(* PLC project CookiePLC, Unknown Unnamed 1 *)
(* stored: creationDateTime 2025-02-05T12:34:47, modificationDateTime 2025-11-16T22:54:03 *)

FUNCTION_BLOCK mixer_rpm_function
  VAR_OUTPUT
    output_rpm : WORD;
  END_VAR
  VAR_INPUT
    valve_status : BOOL;
    hopper_weight : REAL;
    mixer_status : BOOL;
  END_VAR
  VAR
    noise : INT;
  END_VAR
  VAR_IN_OUT
    counter : INT;
  END_VAR

            counter := counter + 1;
IF counter > 10000 THEN
  counter := 0;
END_IF;

noise := counter MOD 2;

IF hopper_weight = 0.0 AND mixer_status = 1 THEN
  output_rpm := INT_TO_WORD(70 + noise);
ELSIF hopper_weight > 0.0 AND mixer_status = 1 AND valve_status = 1 THEN
  output_rpm := INT_TO_WORD(35 + noise);
ELSE
  output_rpm := INT_TO_WORD(0);
END_IF;
          
END_FUNCTION_BLOCK

FUNCTION_BLOCK vacuum_rpm_function
  VAR_INPUT
    input_rpm : WORD;
    vacuum_status : BOOL;
  END_VAR
  VAR_OUTPUT
    output_rpm : WORD;
  END_VAR
  VAR_INPUT
    max_rpm : WORD;
    manual : BOOL := 0;
    dv : BOOL;
  END_VAR
  VAR
    noise : INT;
  END_VAR
  VAR_IN_OUT
    counter : INT;
  END_VAR

            counter := counter + 1;
IF counter > 10000 THEN
  counter := 0;
END_IF;

noise := counter MOD 5;

IF NOT vacuum_status THEN
  output_rpm := 0;
ELSIF input_rpm > max_rpm THEN
  output_rpm := INT_TO_WORD(WORD_TO_INT(max_rpm) + noise);
ELSIF dv = 1 AND manual = 0 THEN
  output_rpm := INT_TO_WORD(1380 + noise);
ELSIF dv = 0 AND manual = 0 THEN
  output_rpm := INT_TO_WORD(1980 + noise);
ELSE
  IF (counter MOD 2) = 1 THEN
    output_rpm := INT_TO_WORD(WORD_TO_INT(input_rpm) + noise);
  ELSE
    output_rpm := INT_TO_WORD(WORD_TO_INT(input_rpm) - noise);
    END_IF;
END_IF;
          
END_FUNCTION_BLOCK

FUNCTION_BLOCK real_to_words
  VAR_INPUT
    Input : REAL;
  END_VAR
  VAR_OUTPUT
    High : WORD;
    Low : WORD;
  END_VAR

            {
    IEC_REAL var_in;
    IEC_WORD var_out[2];
    
    var_in = GetFbVar(INPUT);
    memcpy(var_out, &var_in, sizeof(var_in));
    SetFbVar(HIGH, var_out[0]);
    SetFbVar(LOW, var_out[1]);
}
    
    
          
END_FUNCTION_BLOCK

FUNCTION_BLOCK words_to_real
  VAR_INPUT
    High : WORD;
    Low : WORD;
  END_VAR
  VAR_OUTPUT
    Result : REAL;
  END_VAR

            {
    IEC_WORD var_in[2];

    IEC_REAL var_out;

    var_in[0] = GetFbVar(HIGH);

    var_in[1] = GetFbVar(LOW);

    memcpy(&var_out, var_in, sizeof(var_out));

    SetFbVar(RESULT, var_out);
}
          
END_FUNCTION_BLOCK

FUNCTION_BLOCK conveyor_fpm_function
  VAR_INPUT
    wirecut_cpm : WORD;
    cookie_margin : REAL;
    cookie_diameter : REAL;
  END_VAR
  VAR_OUTPUT
    conveyor_fpm : REAL;
  END_VAR

            conveyor_fpm := (WORD_TO_REAL(wirecut_cpm) * (cookie_margin+cookie_diameter)) / 12.0;
          
END_FUNCTION_BLOCK

FUNCTION_BLOCK flour_alarm_check
  VAR_INPUT
    Flour_weight : REAL;
  END_VAR
  VAR_OUTPUT
    Alarm : BOOL := FALSE;
  END_VAR

            IF Flour_weight <= 100.0 THEN
  Alarm := TRUE;
ELSE
  Alarm := FALSE;
END_IF;

          
END_FUNCTION_BLOCK

FUNCTION_BLOCK hopper_alarm_check
  VAR_INPUT
    Hopper_weight : REAL;
  END_VAR
  VAR_OUTPUT
    Alarm : BOOL := FALSE;
  END_VAR

            IF Hopper_weight <= 10.0 THEN
  Alarm := TRUE;
ELSE
  Alarm := FALSE;
END_IF;

          
END_FUNCTION_BLOCK

FUNCTION_BLOCK papercutter_cpm_function
  VAR
    rows : REAL;
  END_VAR
  VAR_INPUT
    paper_cutter : BOOL;
    cookie_diameter : REAL;
    cookie_margin : REAL;
    conveyor_fpm : REAL;
  END_VAR
  VAR
    float_cpm : REAL;
  END_VAR
  VAR_OUTPUT
    papercut_cpm : WORD;
  END_VAR

            
IF paper_cutter THEN
  rows := 5.0;
  float_cpm := (conveyor_fpm * 12.0) / (rows * (cookie_diameter+cookie_margin));
  papercut_cpm := REAL_TO_WORD(float_cpm);
ELSE
  papercut_cpm := 0;
END_IF;
          
END_FUNCTION_BLOCK

FUNCTION_BLOCK sugar_alarm_check
  VAR_INPUT
    Sugar_weight : REAL;
  END_VAR
  VAR_OUTPUT
    Alarm : BOOL := FALSE;
  END_VAR

            IF Sugar_weight <= 100.0 THEN
  Alarm := TRUE;
ELSE
  Alarm := FALSE;
END_IF;

          
END_FUNCTION_BLOCK

FUNCTION_BLOCK vacuum_alarm_rpm
  VAR_INPUT
    Dv : BOOL;
  END_VAR
  VAR_OUTPUT
    Cfm : REAL;
  END_VAR
  VAR_INPUT
    Vacuum_rpm : WORD;
  END_VAR
  VAR_OUTPUT
    Alarm : BOOL := FALSE;
  END_VAR

            

Cfm := ((-1.275 * 0.0000001) * (WORD_TO_REAL(Vacuum_rpm) * WORD_TO_REAL(Vacuum_rpm)) + (0.7896 * WORD_TO_REAL(Vacuum_rpm)) - 365.43);

IF Dv = 1 AND Cfm < 687.0 THEN 
  Alarm := TRUE;
ELSIF Dv = 0 AND Cfm < 1178.0 THEN
  Alarm := TRUE;
ELSE
  Alarm := FALSE;
END_IF;
  
          
END_FUNCTION_BLOCK

FUNCTION_BLOCK wirecut_cpm_function
  VAR_IN_OUT
    wirecut_cpm : WORD;
  END_VAR
  VAR_INPUT
    wirecutter : BOOL;
  END_VAR

            IF wirecutter THEN
  wirecut_cpm := 200;
ELSE
  wirecut_cpm := 0;
END_IF;
          
END_FUNCTION_BLOCK

PROGRAM tag_display
  VAR
    lcs_1_low AT %QW100 : WORD;  (* Load cell 1 for sugar (lower integer) *)
    lcs_1_high AT %QW101 : WORD;  (* Load cell 1 for sugar (higher integer) *)
    lcs_2_low AT %QW102 : WORD;  (* Load cell 2 for sugar (lower integer) *)
    lcs_2_high AT %QW103 : WORD;  (* Load cell 2 for sugar (higher integer) *)
    lcs_3_low AT %QW104 : WORD;  (* Load cell 3 for sugar (lower integer) *)
    lcs_3_high AT %QW105 : WORD;  (* Load cell 3 for sugar (higher integer) *)
    lcs_4_low AT %QW106 : WORD;  (* Load cell 4 for sugar (lower integer) *)
    lcs_4_high AT %QW107 : WORD;  (* Load cell 4 for sugar (higher integer) *)
    lcf_1_low AT %QW108 : WORD;  (* Load cell 1 for flour (lower integer) *)
    lcf_1_high AT %QW109 : WORD;  (* Load cell 1 for flour (higher integer) *)
    lcf_2_low AT %QW110 : WORD;  (* Load cell 2 for flour (lower integer) *)
    lcf_2_high AT %QW111 : WORD;  (* Load cell 2 for flour (higher integer) *)
    lcf_3_low AT %QW112 : WORD;  (* Load cell 3 for flour (lower integer) *)
    lcf_3_high AT %QW113 : WORD;  (* Load cell 3 for flour (higher integer) *)
    lcf_4_low AT %QW114 : WORD;  (* Load cell 4 for flour (lower integer) *)
    lcf_4_high AT %QW115 : WORD;  (* Load cell 4 for flour (higher integer) *)
    lch_high AT %QW99 : WORD;  (* Load cell for hopper (higher integer) *)
    lch_low AT %QW98 : WORD;  (* Load cell for hopper (lower integer) *)
    lcm_high AT %QW97 : WORD;  (* Load cell for mixer (higher integer) *)
    lcm_low AT %QW96 : WORD;  (* Load cell for mixer (lower integer) *)
    trough_weight_high AT %QW95 : WORD;  (* Weight for trough (higher integer) *)
    trough_weight_low AT %QW94 : WORD;  (* Weight for trough (lower integer) *)
    vacuum_rpm AT %QW1001 : WORD;  (* Vacuum RPM *)
    mixer_rpm AT %QW1003 : WORD;  (* Mixer RPM *)
    wirecut_cpm AT %QW1006 : WORD := 0;  (* Wirecut cuts per minute *)
    papercut_cpm AT %QW1009 : WORD;  (* Papercutter cuts per minute *)
    conveyor_fpm AT %MD13 : REAL;  (* Conveyor feet per minute *)
    conveyor_fpm_high AT %QW121 : WORD := 0;  (* Conveyor feet per minute (high integer) *)
    conveyor_fpm_low AT %QW120 : WORD := 0;  (* Conveyor feet per minute (low integer) *)
    lcs_1 AT %MD0 : REAL;  (* Load cell 1 for sugar (combined float) *)
    lcs_2 AT %MD1 : REAL;  (* Load cell 2 for sugar (combined float) *)
    lcs_3 AT %MD2 : REAL;  (* Load cell 3 for sugar (combined float) *)
    lcs_4 AT %MD3 : REAL;  (* Load cell 4 for sugar (combined float) *)
    lcf_1 AT %MD4 : REAL;  (* Load cell 1 for flour (combined float) *)
    lcf_2 AT %MD5 : REAL;  (* Load cell 2 for flour (combined float) *)
    lcf_3 AT %MD6 : REAL;  (* Load cell 3 for flour (combined float) *)
    lcf_4 AT %MD7 : REAL;  (* Load cell 4 for flour (combined float) *)
    lch AT %MD8 : REAL := 0.0;  (* Load cell for hopper (combined float) *)
    lcm AT %MD11 : REAL := 0.0;  (* Load cell for mixer (combined float) *)
    trough_weight AT %MD12 : REAL := 0.0;  (* Trough weight (combined float) *)
    flour_weight AT %MD9 : REAL := 0.0;  (* Flour weight (combined float) *)
    flour_weight_high AT %QW117 : WORD;  (* Flour weight (higher integer) *)
    flour_weight_low AT %QW116 : WORD;  (* Flour weight (lower integer) *)
    sugar_weight AT %MD10 : REAL := 0.0;  (* Sugar weight (combined float) *)
    sugar_weight_high AT %QW219 : WORD;  (* Sugar weight (higher integer) *)
    sugar_weight_low AT %QW218 : WORD;  (* Sugar weight (lower integer) *)
    tunnel_temp AT %MD15 : REAL;  (* Tunnel temperature *)
    tunnel_temp_high AT %QW303 : WORD := 0;  (* Tunnel temperature (higher integer) *)
    tunnel_temp_low AT %QW302 : WORD := 0;  (* Tunnel temperature (lower integer) *)
    nitrogen_volume AT %MD14 : REAL;  (* Volume of nitrogen *)
    nitrogen_volume_high AT %QW301 : WORD := 0;  (* Volume of nitrogen (higher integer) *)
    nitrogen_volume_low AT %QW300 : WORD := 0;  (* Volume of nitrogen (lower integer) *)
    rv_1 AT %QX87.4 : BOOL;  (* Rotary valve 1 (flour) *)
    rv_2 AT %QX87.5 : BOOL;  (* Rotary valve 2 (sugar) *)
    rv_3 AT %QX87.6 : BOOL;  (* Rotary valve 3 (hopper) *)
    dv AT %QX87.7 : BOOL;  (* Diverter valve *)
    vacuum AT %QX88.0 : BOOL;  (* Vacuum on state *)
    mixer AT %QX88.1 : BOOL;  (* Mixer on state *)
    flour_alarm AT %QX88.2 : BOOL := false;  (* Flour alarm (if flour_weight<1000) *)
    sugar_alarm AT %QX88.3 : BOOL := false;  (* Sugar alarm (if sugar_weight<1000) *)
    hopper_alarm AT %QX88.4 : BOOL := false;  (* Hopper alarm (if lch<100) *)
    vacuum_alarm AT %QX88.5 : BOOL := false;  (* Vacuum alarm *)
    vacuum_manual AT %QX88.6 : BOOL := false;  (* Vacuum manual control state *)
    wirecutter AT %QX88.7 : BOOL := false;  (* Wirecutter on state *)
    trough_transfer AT %QX89.1 : BOOL := false;  (* Trough transfer state *)
    conveyor AT %QX89.4 : BOOL := true;  (* Conveyor on state *)
    paper_cutter AT %QX89.5 : BOOL := false;  (* Papercutter on state *)
    gv_1 AT %QX89.6 : BOOL := false;  (* Gate valve 1 (nitrogen) *)
    fan_1 AT %QX89.7 : BOOL := false;  (* Fan 1 (nitrogen tunnel) *)
    fan_2 AT %QX90.0 : BOOL := false;  (* Fan 2 (nitrogen tunnel) *)
    fan_3 AT %QX90.1 : BOOL := false;  (* Fan 3 (nitrogen tunnel) *)
    exhaust_fan AT %QX90.2 : BOOL := false;  (* Exhaust fan (nitrogen tunnel) *)
    CFM AT %MD20 : REAL;  (* Calculated cubic feet per minute of material *)
    reset AT %QX125.0 : BOOL := false;  (* Restart option for simulation *)
  END_VAR
  VAR
    words_to_real0 : words_to_real;
    words_to_real1 : words_to_real;
    words_to_real2 : words_to_real;
    words_to_real3 : words_to_real;
    words_to_real4 : words_to_real;
    words_to_real5 : words_to_real;
    words_to_real6 : words_to_real;
    words_to_real7 : words_to_real;
    words_to_real8 : words_to_real;
    flour_alarm_check0 : flour_alarm_check;
    sugar_alarm_check0 : sugar_alarm_check;
    hopper_alarm_check0 : hopper_alarm_check;
    vacuum_alarm_rpm0 : vacuum_alarm_rpm;
    real_to_words0 : real_to_words;
    real_to_words1 : real_to_words;
    vacuum_max_rpm : WORD := 3600;  (* Max rpm of vacuum *)
    mixer_max_rpm : WORD := 80;  (* Max rpm of mixer *)
    mixer_rpm_function0 : mixer_rpm_function;
    vacuum_rpm_function0 : vacuum_rpm_function;
    cookie_diameter : REAL := 1.5;  (* Diameter of individual cookies (in) *)
    cookie_margin : REAL := 0.5;  (* Margin between cookies on paper (in) *)
    papercutter_cpm_function0 : papercutter_cpm_function;
    conveyor_fpm_function0 : conveyor_fpm_function;
    words_to_real9 : words_to_real;
    words_to_real10 : words_to_real;
    real_to_words2 : real_to_words;
    wirecut_cpm_function0 : wirecut_cpm_function;
    words_to_real11 : words_to_real;
    words_to_real12 : words_to_real;
  END_VAR
  VAR
    box_maker AT %QX90.3 : BOOL := false;  (* Box maker on state *)
    taper AT %QX90.4 : BOOL := false;  (* Taper on state *)
    labeler AT %QX90.5 : BOOL := false;  (* Labeler on state *)
    palletizer AT %QX90.6 : BOOL := false;  (* Palletizer on state *)
    palletizer_grabbing AT %QX90.7 : BOOL := false;  (* Palletizer grabbing state *)
    wrapper AT %QX91.0 : BOOL := false;  (* Wrapper on state *)
    wrapper_conveying AT %QX91.1 : BOOL := false;  (* Wrapper conveyor on state *)
    conveyor_1 AT %QX91.2 : BOOL := true;  (* Conveyor 1 on state *)
    conveyor_2 AT %QX91.3 : BOOL := true;  (* Conveyor 2 on state *)
    conveyor_3 AT %QX91.4 : BOOL := true;  (* Conveyor 3 on state *)
    conveyor_4 AT %QX91.5 : BOOL := true;  (* Conveyor 4 on state *)
    conveyor_5 AT %QX91.6 : BOOL := true;  (* Conveyor 5 on state *)
    ps_1 AT %QX91.7 : BOOL := false;  (* Photoelectric sensor 1 *)
    ps_2 AT %QX92.0 : BOOL := false;  (* Photoelectric sensor 2 *)
    ps_3 AT %QX92.1 : BOOL := false;  (* Photoelectric sensor 3 *)
    ps_4 AT %QX92.2 : BOOL := false;  (* Photoelectric sensor 4 *)
    ps_5 AT %QX92.3 : BOOL := false;  (* Photoelectric sensor 5 *)
    ps_6 AT %QX92.4 : BOOL := false;  (* Photoelectric sensor 6 *)
    bagger AT %QX92.5 : BOOL := false;  (* Bagger on state *)
    palletizer_rotation AT %QW1012 : INT := 180;  (* Palletizer arm position 1, 2 , or 3 *)
    box_count AT %QW1013 : INT := 0;  (* Number of boxes on the wrapper *)
    wrapper_wrapping AT %QX92.6 : BOOL := false;  (* True if the wrapper is currently wrapping *)
    boxing AT %QX92.7 : BOOL := false;  (* True if the boxer is currently boxing *)
    taping AT %QX93.0 : BOOL := false;  (* True if the taper is currently taping *)
    conveying_1 AT %QX93.1 : BOOL := false;  (* True if conveyor_1 is currently conveying *)
    conveying_2 AT %QX93.2 : BOOL := false;  (* True if conveyor_2 is currently conveying *)
    conveying_3 AT %QX93.3 : BOOL := false;  (* True if conveyor_3 is currently conveying *)
    conveying_4 AT %QX93.4 : BOOL := false;  (* True if conveyor_4 is currently conveying *)
    conveying_5 AT %QX93.5 : BOOL := false;  (* True if conveyor_5 is currently conveying *)
    palletizer_moving AT %QX93.6 : BOOL := false;  (* True if the palletizer arm is moving *)
    bagging AT %QX93.7 : BOOL := false;  (* Set to true if the bagger is bagging *)
    machine_1 AT %QW500 : INT := 0;  (* State value for state machine 1 *)
    machine_2 AT %QW501 : INT := 0;  (* State value for state machine 2 *)
    machine_3 AT %QW502 : INT := 0;  (* State value for state machine 3 *)
    machine_4 AT %QW503 : INT := 0;  (* State value for state machine 4 *)
  END_VAR
  VAR
    state_0 : INT := 0;  (* State constant *)
    state_1 : INT := 1;  (* State constant *)
    state_2 : INT := 2;  (* State constant *)
    state_3 : INT := 3;  (* State constant *)
    state_4 : INT := 4;  (* State constant *)
    state_5 : INT := 5;  (* State constant *)
    state_6 : INT := 6;  (* State constant *)
    pos_1 : INT := 225;  (* Palletizer rotation constant (degrees) *)
    pos_2 : INT := 180;  (* Palletizer rotation constant (degrees) *)
    pos_3 : INT := 130;  (* Palletizer rotation constant (degrees) *)
  END_VAR
  VAR
    roe_1 AT %QX94.0 : BOOL := false;  (* Sensor for palletizer pos_1 *)
    roe_2 AT %QX94.1 : BOOL := false;  (* Sensor for palletizer pos_2 *)
    roe_3 AT %QX94.2 : BOOL := false;  (* Sensor for palletizer pos_3 *)
    add_ingredients AT %QX94.3 : BOOL := false;  (* Coil for adding additional non-bulk ingredients *)
  END_VAR
  VAR  (* added by the conversion: wires and edge detectors of the diagram *)
    _EQ264_OUT : BOOL;
  END_VAR

(* LD diagram, written out as Structured Text *)
words_to_real0(High := lcf_1_high, Low := lcf_1_low);
lcf_1 := words_to_real0.Result;
words_to_real1(High := lcf_2_high, Low := lcf_2_low);
lcf_2 := words_to_real1.Result;
words_to_real2(High := lcf_3_high, Low := lcf_3_low);
lcf_3 := words_to_real2.Result;
words_to_real3(High := lcf_4_high, Low := lcf_4_low);
lcf_4 := words_to_real3.Result;
words_to_real4(High := lcs_1_high, Low := lcs_1_low);
lcs_1 := words_to_real4.Result;
words_to_real5(High := lcs_2_high, Low := lcs_2_low);
lcs_2 := words_to_real5.Result;
words_to_real6(High := lcs_3_high, Low := lcs_3_low);
lcs_3 := words_to_real6.Result;
words_to_real7(High := lcs_4_high, Low := lcs_4_low);
lcs_4 := words_to_real7.Result;
flour_weight := lcf_1 + lcf_2 + (lcf_3 + lcf_4);
flour_alarm_check0(Flour_weight := flour_weight);
flour_alarm := flour_alarm_check0.Alarm;
sugar_weight := lcs_1 + lcs_2 + (lcs_3 + lcs_4);
words_to_real8(High := lch_high, Low := lch_low);
lch := words_to_real8.Result;
hopper_alarm_check0(Hopper_weight := lch);
hopper_alarm := hopper_alarm_check0.Alarm;
vacuum_alarm_rpm0(Dv := dv, Vacuum_rpm := vacuum_rpm);
vacuum_alarm := vacuum_alarm_rpm0.Alarm;
CFM := vacuum_alarm_rpm0.Cfm;
real_to_words0(Input := flour_weight);
flour_weight_high := real_to_words0.High;
flour_weight_low := real_to_words0.Low;
real_to_words1(Input := sugar_weight);
sugar_weight_high := real_to_words1.High;
sugar_weight_low := real_to_words1.Low;
sugar_alarm_check0(Sugar_weight := sugar_weight);
sugar_alarm := sugar_alarm_check0.Alarm;
mixer_rpm_function0(valve_status := rv_3, hopper_weight := lch, mixer_status := mixer, counter := mixer_rpm_function0.counter);
mixer_rpm := mixer_rpm_function0.output_rpm;
vacuum_rpm_function0(input_rpm := vacuum_rpm, vacuum_status := vacuum, max_rpm := vacuum_max_rpm, manual := vacuum_manual, dv := dv, counter := vacuum_rpm_function0.counter);
vacuum_rpm := vacuum_rpm_function0.output_rpm;
words_to_real9(High := trough_weight_high, Low := trough_weight_low);
trough_weight := words_to_real9.Result;
words_to_real10(High := lcm_high, Low := lcm_low);
lcm := words_to_real10.Result;
papercutter_cpm_function0(paper_cutter := paper_cutter, cookie_diameter := cookie_diameter, cookie_margin := cookie_margin, conveyor_fpm := conveyor_fpm);
papercut_cpm := papercutter_cpm_function0.papercut_cpm;
conveyor_fpm_function0(wirecut_cpm := wirecut_cpm, cookie_margin := cookie_margin, cookie_diameter := cookie_diameter);
conveyor_fpm := conveyor_fpm_function0.conveyor_fpm;
real_to_words2(Input := conveyor_fpm);
conveyor_fpm_high := real_to_words2.High;
conveyor_fpm_low := real_to_words2.Low;
wirecut_cpm_function0(wirecut_cpm := wirecut_cpm, wirecutter := wirecutter);
wirecut_cpm := wirecut_cpm_function0.wirecut_cpm;
words_to_real11(High := nitrogen_volume_high, Low := nitrogen_volume_low);
nitrogen_volume := words_to_real11.Result;
words_to_real12(High := tunnel_temp_high, Low := tunnel_temp_low);
tunnel_temp := words_to_real12.Result;
(* First state of the third state machine, if ps_5 is set to true and palletizer is on and not grabbing/moving, set palletizer_moving to true *)
(* First state of the first state machine, start boxing if the box maker is on. *)
(* First state of the second state machine, set conveying_3 to true if ps_3 is true and conveyor_3 is on. *)
(* First state of the fourth state machine, set wrapper_wrapping to true if the wrapper is on, there's no pallet at the end of the conveyor (ps_6 is false) and the box count is equal to 40. *)
IF machine_1 = state_0 AND box_maker THEN boxing := TRUE; END_IF;
IF machine_1 = state_0 AND box_maker THEN machine_1 := state_1; END_IF;
(* Second state of the first state machine, if the box maker is done boxing and the conveyor 1 is on, set conveying_1 to true. *)
(* Second state of the second state machine, if ps_4 is true, and taper is on, set taping to true. *)
IF machine_1 = state_1 AND NOT boxing AND conveyor_1 THEN conveying_1 := TRUE; END_IF;
IF machine_1 = state_1 AND NOT boxing AND conveyor_1 THEN machine_1 := state_2; END_IF;
(* Second state of the fourth state machine, set wrapper_conveying to true if the wrapper is on and it is done wrapping. *)
(* Second state of the third state machine, if roe_1 is set to true then set palletizer_moving to false *)
(* Thrid state of the first state machine, if the ps_1 is on and bagger is on, set conveying_1 to false and set bagging to true. *)
(* Third (and final) state of the second state machine, if taping is false and conveyor_4 is on set conveying_4 to true. *)
IF machine_1 = state_2 AND ps_1 AND bagger THEN bagging := TRUE; END_IF;
IF machine_1 = state_2 AND ps_1 AND bagger THEN machine_1 := state_3; END_IF;
(* Third state of the third state machine, set palletizer_rotation to 225, palletizer_grabbing to true, and palletizer_moving to true if the palletizer is on. *)
(* Third state of the fourth state machine, set conveying_4 to true if wrapper_conveying is false and conveyor_4 is on. *)
(* Fourth state of the first state machine, if the bagger is done bagging and conveyor_2 is on, set conveying_2 to true. *)
(* Fourth state of the fourth state machine, if ps_6 is on conveying_5 is set to false. *)
IF machine_1 = state_3 AND conveyor_2 AND NOT bagging THEN machine_1 := state_4; END_IF;
IF machine_1 = state_3 AND conveyor_2 AND NOT bagging THEN conveying_2 := TRUE; END_IF;
(* Fifth state of the first state machine, if ps_2 is on conveying_2 is set to false. *)
(* Fourth state of the third state machine, if roe_2 is set to true then set palletizer_moving to false *)
(* Sixth (and final) state of the first state machine, if ps_2 is false move back to start state. *)
IF machine_1 = state_5 AND NOT ps_2 THEN machine_1 := state_0; END_IF;
IF machine_2 = state_0 AND conveyor_3 AND ps_3 THEN conveying_3 := TRUE; END_IF;
IF machine_2 = state_0 AND conveyor_3 AND ps_3 THEN machine_2 := state_1; END_IF;
IF machine_2 = state_1 AND ps_4 AND taper THEN taping := TRUE; END_IF;
IF machine_2 = state_1 AND ps_4 AND taper THEN machine_2 := state_2; END_IF;
IF machine_2 = state_2 AND NOT ps_5 AND NOT taping AND conveyor_4 THEN conveying_4 := TRUE; END_IF;
IF machine_2 = state_2 AND NOT ps_5 AND NOT taping AND conveyor_4 THEN machine_2 := state_0; END_IF;
IF machine_3 = state_2 AND palletizer THEN machine_3 := state_3; END_IF;
IF machine_3 = state_2 AND palletizer THEN palletizer_moving := TRUE; END_IF;
(* Fifth state of the third state machine. Set palletizer_rotation to 130 and palletizer_moving to true if wrapper_wrapping, wrapper_conveying are false, and palletizer is true. *)
IF machine_3 = state_4 AND palletizer AND NOT wrapper_conveying AND NOT wrapper_wrapping THEN palletizer_moving := TRUE; END_IF;
IF machine_3 = state_4 AND palletizer AND NOT wrapper_conveying AND NOT wrapper_wrapping THEN machine_3 := state_5; END_IF;
IF machine_3 = state_2 AND palletizer THEN palletizer_rotation := pos_2; END_IF;
(* Sixth state of the third state machine, if roe_3 is set to true then set palletizer_moving to false *)
(* Seventh state of the third state machine, set palletizer_rotation to 180 degrees, palletizer_moving to true, palletizer_grabbing to false, and add 1 to the box count if palletizer is true. *)
_EQ264_OUT := machine_3 = state_6;
IF _EQ264_OUT THEN palletizer_rotation := pos_2; END_IF;
IF _EQ264_OUT AND palletizer THEN box_count := box_count + 1; END_IF;
IF _EQ264_OUT AND palletizer THEN machine_3 := state_3; END_IF;
IF machine_4 = state_0 AND box_count >= 10 AND wrapper AND NOT ps_6 THEN wrapper_wrapping := TRUE; END_IF;
IF machine_3 = state_0 AND ps_5 AND NOT palletizer_grabbing AND palletizer THEN machine_3 := state_1; END_IF;
IF machine_4 = state_1 AND wrapper AND NOT wrapper_wrapping THEN wrapper_conveying := TRUE; END_IF;
IF machine_4 = state_0 AND box_count >= 10 AND wrapper AND NOT ps_6 THEN machine_4 := state_1; END_IF;
IF machine_4 = state_1 AND wrapper AND NOT wrapper_wrapping THEN machine_4 := state_2; END_IF;
IF machine_4 = state_2 AND conveyor_5 AND NOT wrapper_conveying THEN conveying_5 := TRUE; END_IF;
IF machine_4 = state_2 AND conveyor_5 AND NOT wrapper_conveying THEN machine_4 := state_3; END_IF;
IF _EQ264_OUT AND palletizer THEN palletizer_grabbing := FALSE; END_IF;
IF _EQ264_OUT AND palletizer THEN palletizer_moving := TRUE; END_IF;
IF machine_1 = state_2 AND ps_1 THEN conveying_1 := FALSE; END_IF;
IF machine_1 = state_4 AND ps_2 THEN machine_1 := state_5; END_IF;
IF machine_1 = state_4 AND ps_2 THEN conveying_2 := FALSE; END_IF;
IF machine_2 = state_1 AND ps_4 THEN conveying_3 := FALSE; END_IF;
IF machine_3 = state_0 AND ps_5 THEN conveying_4 := FALSE; END_IF;
IF machine_4 = state_3 AND ps_6 THEN machine_4 := state_0; END_IF;
IF machine_4 = state_3 AND ps_6 THEN conveying_5 := FALSE; END_IF;
IF machine_3 = state_0 AND ps_5 AND NOT palletizer_grabbing AND palletizer THEN palletizer_moving := TRUE; END_IF;
IF machine_3 = state_0 AND ps_5 AND NOT palletizer_grabbing AND palletizer THEN palletizer_rotation := pos_1; END_IF;
IF machine_3 = state_1 AND roe_1 THEN palletizer_moving := FALSE; END_IF;
IF machine_3 = state_3 AND roe_2 AND palletizer_grabbing THEN machine_3 := state_4; END_IF;
IF machine_3 = state_3 AND roe_2 THEN palletizer_moving := FALSE; END_IF;
IF machine_3 = state_4 AND palletizer AND NOT wrapper_conveying AND NOT wrapper_wrapping THEN palletizer_rotation := pos_3; END_IF;
IF machine_3 = state_5 AND roe_3 THEN machine_3 := state_6; END_IF;
IF machine_3 = state_5 AND roe_3 THEN palletizer_moving := FALSE; END_IF;
IF machine_3 = state_3 AND roe_2 AND NOT palletizer_grabbing THEN machine_3 := state_0; END_IF;
IF machine_3 = state_1 AND roe_1 THEN machine_3 := state_2; END_IF;
IF machine_3 = state_0 AND ps_5 AND NOT palletizer_grabbing AND palletizer THEN palletizer_grabbing := TRUE; END_IF;
IF machine_4 = state_0 AND box_count >= 10 AND wrapper AND NOT ps_6 THEN box_count := 0; END_IF;
END_PROGRAM

FUNCTION_BLOCK wirecut_ppm_function
  VAR_INPUT
    wirecut_cpm : WORD;
  END_VAR
  VAR
    cookie_weight : REAL;
    cookie_count : REAL;
  END_VAR
  VAR_OUTPUT
    wirecut_ppm : REAL;
  END_VAR

            cookie_count := 8.0;
cookie_weight := 0.3;
wirecut_ppm := (WORD_TO_REAL(wirecut_cpm) * cookie_count * cookie_weight)/16.0;
          
END_FUNCTION_BLOCK

CONFIGURATION Config0
  RESOURCE Res0 ON PLC
    TASK task0(INTERVAL := T#20ms, PRIORITY := 0);
    PROGRAM instance0 WITH task0 : tag_display;
  END_RESOURCE
END_CONFIGURATION
